# B&R Automation Studio project Lecture_08_jbl
Automation Studio 4.8.2.72

## Configuration Config1

### Task classes (Cpu.sw)
```
Cyclic#4:
  Assignment <- Assignment1.prg
  Program <- (binary)
  Assignmen1 <- Assignment2.prg
  Assignmen2 <- Assignment2_if.prg
Binaries: udbdef, FWRules, TCData, sysconf, Role, User, iomap, ashwd, asfw, arconfig, ashwac
Libraries: runtime, astime, asieccon
```

### Hardware
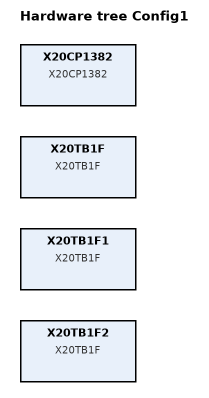
```
X20CP1382 : X20CP1382 v1.10.0.0  [X1 -> X1.SL; X2 -> X2.SL; X3 -> X3.SL]
  Module X1 (Type=X1, Virtual=true, Version=1.10.0.0)
    Connection (Connector=SS1, TargetModule=X20TB1F, TargetConnector=SS)
    Connection (Connector=SL, TargetModule=X20CP1382, TargetConnector=X1)
  Module X2 (Type=X2, Virtual=true, Version=1.10.0.0)
    Connection (Connector=SS1, TargetModule=X20TB1F1, TargetConnector=SS)
    Connection (Connector=SL, TargetModule=X20CP1382, TargetConnector=X2)
  Module X3 (Type=X3, Virtual=true, Version=1.10.0.0)
    Connection (Connector=SS1, TargetModule=X20TB1F2, TargetConnector=SS)
    Connection (Connector=SL, TargetModule=X20CP1382, TargetConnector=X3)
  Connector IF2:
    ActivateDevice = 1
  ConfigurationID = Lecture_08_jbl_Config1
  Simulation = 1
X20TB1F : X20TB1F v1.0.0.0
X20TB1F1 : X20TB1F v1.0.0.0
X20TB1F2 : X20TB1F v1.0.0.0
```

## Logical view

### Program Logical/Assignment1 (IEC)

#### Variables.var
```iecst
VAR
	old_input : BOOL;
	input : BOOL;
	falling_edge : BOOL;
END_VAR
```

#### Main.st
```iecst
PROGRAM _INIT
	(* Insert code here *)
	falling_edge := FALSE;

END_PROGRAM

PROGRAM _CYCLIC
	(* Insert code here *)

	IF input = TRUE THEN
		old_input := FALSE;
	ELSE
		old_input := TRUE;
	END_IF;

	IF input = FALSE AND old_input = TRUE THEN
		falling_edge := TRUE;
	ELSE
		falling_edge := FALSE;
	END_IF

END_PROGRAM

PROGRAM _EXIT
	(* Insert code here *)

END_PROGRAM
```

### Program Logical/Assignment2 (IEC)

#### Main.st
```iecst
PROGRAM _INIT
	(* Insert code here *)

END_PROGRAM

PROGRAM _CYCLIC
	(* Insert code here *)

END_PROGRAM

PROGRAM _EXIT
	(* Insert code here *)

END_PROGRAM
```

### Program Logical/Assignment2_if (IEC)

#### Variables.var
```iecst
VAR
	doConvBottom : BOOL;
	doLiftTop : BOOL;
	doLiftBottom : BOOL;
	doLiftUnload : BOOL;
	dooConvTop : BOOL;
	doBoxLift : BOOL;
END_VAR
```

#### Main.st
```iecst
PROGRAM _INIT
	(* Insert code here *)

END_PROGRAM

PROGRAM _CYCLIC
	(* Insert code here *)

	doConvTop := NOT(doConvBottom) AND NOT(doLiftUnload) AND doLiftTop AND NOT(doBoxLift);
	doConvBottom := NOT(doConvTop) AND NOT(doLiftUnload) AND doLiftBottom AND NOT(doBoxLift);

END_PROGRAM

PROGRAM _EXIT
	(* Insert code here *)

END_PROGRAM
```

### Variables.var
```iecst
VAR
	falling_edge : BOOL;
END_VAR
```

Listed in the project but not available here: Logical/Global.typ, Logical/Global.var, Logical/Libraries
